PROGRAM P_AutoMode
VAR
	tonCycle				: TON; //timer implemented to reduce CPU usage
	
	bIsDay			: BOOL := FALSE;
	bIsNight		: BOOL := FALSE;
	
	rtIsDay			: R_TRIG;
	rtIsNight		: R_TRIG;			
	
	ft_arrManual	: ARRAY [1..byStreetLampsCount] OF F_TRIG;
	i				: INT;	//for loop iterator
END_VAR

//init tonCycle
tonCycle(IN:=NOT tonCycle.Q, PT:=T#1S);
//init rising edge detection
rtIsDay(CLK := bIsDay);
rtIsNight(CLK := bIsNight);

//check day-night status every 1S
IF tonCycle.Q THEN
	
	//if it is a night
	IF F_IsNight() THEN
		//set flags accordingly
		bIsNight := TRUE;
		bIsDay := FALSE;
	//else, it is a day
	ELSE
		//set flags accordingly
		bIsNight := FALSE;
		bIsDay := TRUE;
	END_IF

END_IF

//if a night has come
IF rtIsNight.Q THEN
	//turn lights ON
	//if they are not in manual mode	
	IF NOT GVL_IO.arrStreetLamps[1].bManualCtrl  THEN fbBACnet_AV_SL_Level_1.fPV  := c_byBrightness_Night; END_IF
	IF NOT GVL_IO.arrStreetLamps[2].bManualCtrl  THEN fbBACnet_AV_SL_Level_2.fPV  := c_byBrightness_Night; END_IF
	IF NOT GVL_IO.arrStreetLamps[3].bManualCtrl  THEN fbBACnet_AV_SL_Level_3.fPV  := c_byBrightness_Night; END_IF
	IF NOT GVL_IO.arrStreetLamps[4].bManualCtrl  THEN fbBACnet_AV_SL_Level_4.fPV  := c_byBrightness_Night; END_IF
	IF NOT GVL_IO.arrStreetLamps[5].bManualCtrl  THEN fbBACnet_AV_SL_Level_5.fPV  := c_byBrightness_Night; END_IF
	IF NOT GVL_IO.arrStreetLamps[6].bManualCtrl  THEN fbBACnet_AV_SL_Level_6.fPV  := c_byBrightness_Night; END_IF
	IF NOT GVL_IO.arrStreetLamps[7].bManualCtrl  THEN fbBACnet_AV_SL_Level_7.fPV  := c_byBrightness_Night; END_IF
	IF NOT GVL_IO.arrStreetLamps[8].bManualCtrl  THEN fbBACnet_AV_SL_Level_8.fPV  := c_byBrightness_Night; END_IF
	IF NOT GVL_IO.arrStreetLamps[9].bManualCtrl  THEN fbBACnet_AV_SL_Level_9.fPV  := c_byBrightness_Night; END_IF
	IF NOT GVL_IO.arrStreetLamps[10].bManualCtrl THEN fbBACnet_AV_SL_Level_10.fPV := c_byBrightness_Night; END_IF

	//turn one street lamp ON
	GVL_IO.bStreetLamp_DO1 := TRUE;
END_IF

//if a day has come
IF rtIsDay.Q THEN
	//turn all lights OFF
	fbBACnet_AV_SL_Level_1.fPV  := c_byBrightness_Day;
	fbBACnet_AV_SL_Level_2.fPV  := c_byBrightness_Day;
	fbBACnet_AV_SL_Level_3.fPV  := c_byBrightness_Day;
	fbBACnet_AV_SL_Level_4.fPV  := c_byBrightness_Day;
	fbBACnet_AV_SL_Level_5.fPV  := c_byBrightness_Day;
	fbBACnet_AV_SL_Level_6.fPV  := c_byBrightness_Day;
	fbBACnet_AV_SL_Level_7.fPV  := c_byBrightness_Day;
	fbBACnet_AV_SL_Level_8.fPV  := c_byBrightness_Day;
	fbBACnet_AV_SL_Level_9.fPV  := c_byBrightness_Day;
	fbBACnet_AV_SL_Level_10.fPV := c_byBrightness_Day;
	
	//turn one street lamp OFF
	GVL_IO.bStreetLamp_DO1 := FALSE;
	
	//and disable manual mode
	bBACnet_ResetManual := TRUE;
END_IF

//special case - exit manual mode
//when manual mode is turned off
//return brightness level to auto mode level 
FOR i := 1 TO byStreetLampsCount BY 1 DO
	//init falling edge detection
	ft_arrManual[i](CLK := GVL_IO.arrStreetLamps[i].bManualCtrl);
	
	//if manual mode is being turned off
	IF ft_arrManual[i].Q THEN
		//set brightness level to auto mode on this lamp
		//in the night to c_byBrightness_Night
		IF F_IsNight() THEN
			CASE i OF
				1: 	fbBACnet_AV_SL_Level_1.fPV  := c_byBrightness_Night;
				2: 	fbBACnet_AV_SL_Level_2.fPV  := c_byBrightness_Night;
				3: 	fbBACnet_AV_SL_Level_3.fPV  := c_byBrightness_Night;
				4: 	fbBACnet_AV_SL_Level_4.fPV  := c_byBrightness_Night;
				5: 	fbBACnet_AV_SL_Level_5.fPV  := c_byBrightness_Night;
				6: 	fbBACnet_AV_SL_Level_6.fPV  := c_byBrightness_Night;
				7: 	fbBACnet_AV_SL_Level_7.fPV  := c_byBrightness_Night;
				8: 	fbBACnet_AV_SL_Level_8.fPV  := c_byBrightness_Night;
				9: 	fbBACnet_AV_SL_Level_9.fPV  := c_byBrightness_Night;
				10:	fbBACnet_AV_SL_Level_10.fPV := c_byBrightness_Night;
			END_CASE
		ELSE
		//at the daylight to c_byBrightness_Day
			CASE i OF
				1: 	fbBACnet_AV_SL_Level_1.fPV  := c_byBrightness_Day;
				2: 	fbBACnet_AV_SL_Level_2.fPV  := c_byBrightness_Day;
				3: 	fbBACnet_AV_SL_Level_3.fPV  := c_byBrightness_Day;
				4: 	fbBACnet_AV_SL_Level_4.fPV  := c_byBrightness_Day;
				5: 	fbBACnet_AV_SL_Level_5.fPV  := c_byBrightness_Day;
				6: 	fbBACnet_AV_SL_Level_6.fPV  := c_byBrightness_Day;
				7: 	fbBACnet_AV_SL_Level_7.fPV  := c_byBrightness_Day;
				8: 	fbBACnet_AV_SL_Level_8.fPV  := c_byBrightness_Day;
				9: 	fbBACnet_AV_SL_Level_9.fPV  := c_byBrightness_Day;
				10:	fbBACnet_AV_SL_Level_10.fPV := c_byBrightness_Day;
			END_CASE
		END_IF
	END_IF
END_FOR

END_PROGRAM

(* stored: Version 1.1.0.1, ProductVersion 3.1.4024.5
   POU P_AutoMode: Id {3a6df21b-1a42-48ce-9146-75164385b2da}, SpecialFunc None *)
